RoboDK station: TECLADO.rdk

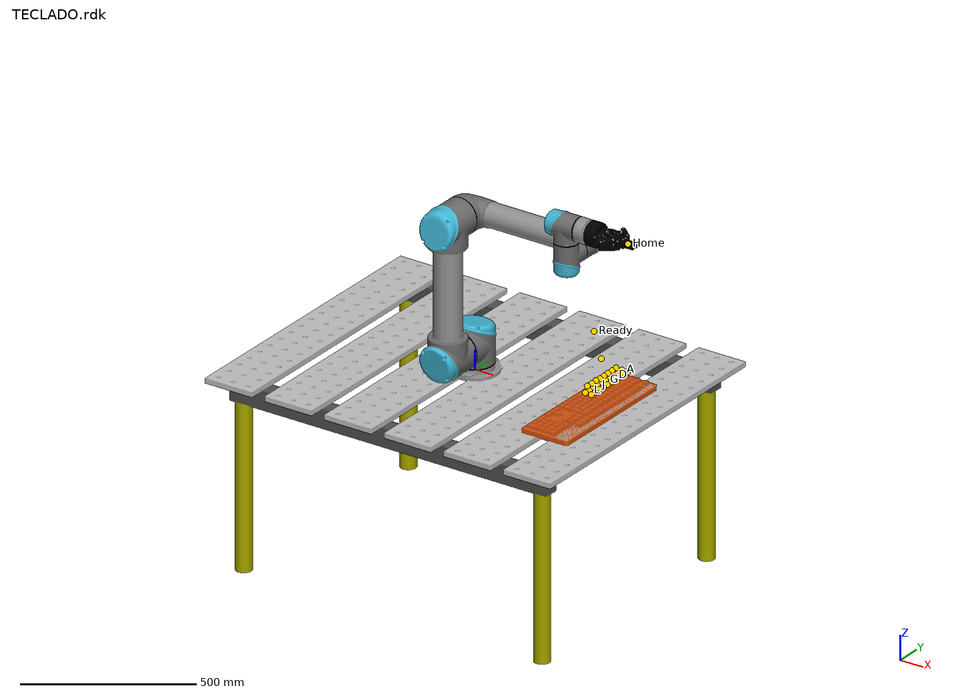
[picture v0: the station drawn from its stored meshes, robots at their saved joint values, targets as dots, program paths as lines]
Station TECLADO (saved by RoboDK 5.5.4). Poses are relative to the parent item; angles as X-Y-Z fixed-axis rotations.
  - frame UR5 Base at (0, 1000, 0) mm
    - robot UR5: 6 axes
        modified DH rows (alpha deg, a mm, theta deg, d mm): 0, 0, 0, 89.2; 90, 0, 180, 0; 0, 425, 0, 0; 0, 392, 0, 109.3; -90, 0, 0, 94.75; 90, 0, 180, 82.5
        joint limits [-360, -360, -360, -360, -360, -360] to [360, 360, 360, 360, 360, 360]; home [0, -90, -90, 0, 90, 0]; saved at [0, -90, -90, 0, 90, 0]
      - tool RobotiQ 2F-85 Gripper (Fully Closed), TCP at (0, 0, 130) mm, size 121.5 x 75 x 160.2 mm
    - object Table 1200x1000mm (Welding) at (0, 0, 0) mm, size 1193.8 x 965.2 x 609.6 mm, geometry from Table-1200x1000mm-Welding (1).sld
    - target Home (Cartesian target) at (604.5, -109.3, 608.95) mm, rotated rx -90 ry 0 rz -90 deg; joints [0, -90, -90, 0, 90, 0] of UR5
    - target Ready (Cartesian target) at (486.75, -109.3, 301.7) mm, rotated rx -180 ry 0 rz -90 deg; joints [0, -90, -90, -90, 90, 0] of UR5
    - target A (Cartesian target) at (400.33, 152.85, 49.84) mm, rotated rx -180 ry 0 rz -90 deg; joints [35.675, -92.543, -127.355, -50.102, 90, 35.675] of UR5
    - target S (Cartesian target) at (400.33, 132.85, 49.84) mm, rotated rx -180 ry 0 rz -90 deg; joints [33.377, -91.633, -128.312, -50.055, 90, 33.377] of UR5
    - target D (Cartesian target) at (400.33, 112.85, 49.84) mm, rotated rx -180 ry 0 rz -90 deg; joints [30.978, -90.828, -129.142, -50.03, 90, 30.978] of UR5
    - target F (Cartesian target) at (400.33, 92.85, 49.84) mm, rotated rx -180 ry 0 rz -90 deg; joints [28.482, -90.138, -129.84, -50.022, 90, 28.482] of UR5
    - target G (Cartesian target) at (400.33, 72.85, 49.84) mm, rotated rx -180 ry 0 rz -90 deg; joints [25.895, -89.569, -130.406, -50.024, 90, 25.895] of UR5
    - target H (Cartesian target) at (400.33, 52.85, 49.84) mm, rotated rx -180 ry 0 rz -90 deg; joints [23.225, -89.131, -130.838, -50.031, 90, 23.225] of UR5
    - target J (Cartesian target) at (400.33, 32.85, 49.84) mm, rotated rx -180 ry 0 rz -90 deg; joints [20.481, -88.828, -131.133, -50.039, 90, 20.481] of UR5
    - target K (Cartesian target) at (400.33, 12.85, 49.84) mm, rotated rx -180 ry 0 rz -90 deg; joints [17.674, -88.666, -131.29, -50.044, 90, 17.674] of UR5
    - target L (Cartesian target) at (400.33, -7.15, 49.84) mm, rotated rx -180 ry 0 rz -90 deg; joints [14.818, -88.645, -131.31, -50.044, 90, 14.818] of UR5
    - target Ñ (Cartesian target) at (400.33, -27.15, 49.84) mm, rotated rx -180 ry 0 rz -90 deg; joints [11.927, -88.768, -131.192, -50.041, 90, 11.927] of UR5
    - target Z (Cartesian target) at (380.33, 152.85, 49.84) mm, rotated rx -180 ry 0 rz -90 deg; joints [37.36, -89.989, -129.989, -50.022, 90, 37.36] of UR5
    - target X (Cartesian target) at (380.33, 132.85, 49.84) mm, rotated rx -180 ry 0 rz -90 deg; joints [34.996, -88.998, -130.968, -50.034, 90, 34.996] of UR5
    - target C (Cartesian target) at (380.33, 112.85, 49.84) mm, rotated rx -180 ry 0 rz -90 deg; joints [32.519, -88.118, -131.817, -50.066, 90, 32.519] of UR5
    - target V (Cartesian target) at (380.33, 92.85, 49.84) mm, rotated rx -180 ry 0 rz -90 deg; joints [29.93, -87.36, -132.533, -50.108, 90, 29.93] of UR5
    - target B (Cartesian target) at (380.33, 72.85, 49.84) mm, rotated rx -180 ry 0 rz -90 deg; joints [27.238, -86.734, -133.112, -50.153, 90, 27.238] of UR5
    - target N (Cartesian target) at (380.33, 52.85, 49.84) mm, rotated rx -180 ry 0 rz -90 deg; joints [24.449, -86.25, -133.555, -50.195, 90, 24.449] of UR5
    - target N (Cartesian target) at (380.33, 32.85, 49.84) mm, rotated rx -180 ry 0 rz -90 deg; joints [21.574, -85.916, -133.857, -50.227, 90, 21.574] of UR5
    - target M (Cartesian target) at (380.33, 12.85, 49.84) mm, rotated rx -180 ry 0 rz -90 deg; joints [18.626, -85.736, -134.019, -50.246, 90, 18.626] of UR5
    - target Q (Cartesian target) at (420.33, 152.85, 49.84) mm, rotated rx -180 ry 0 rz -90 deg; joints [34.128, -95.022, -124.646, -50.332, 90, 34.128] of UR5
    - target W (Cartesian target) at (420.33, 132.85, 49.84) mm, rotated rx -180 ry 0 rz -90 deg; joints [31.895, -94.18, -125.582, -50.237, 90, 31.895] of UR5
    - target E (Cartesian target) at (420.33, 112.85, 49.84) mm, rotated rx -180 ry 0 rz -90 deg; joints [29.573, -93.439, -126.393, -50.168, 90, 29.573] of UR5
    - target R (Cartesian target) at (420.33, 92.85, 49.84) mm, rotated rx -180 ry 0 rz -90 deg; joints [27.165, -92.805, -127.076, -50.119, 90, 27.165] of UR5
    - target T (Cartesian target) at (420.33, 72.85, 49.84) mm, rotated rx -180 ry 0 rz -90 deg; joints [24.678, -92.284, -127.629, -50.086, 90, 24.678] of UR5
    - target Y (Cartesian target) at (420.33, 52.85, 49.84) mm, rotated rx -180 ry 0 rz -90 deg; joints [22.118, -91.884, -128.051, -50.066, 90, 22.118] of UR5
    - target U (Cartesian target) at (420.33, 32.85, 49.84) mm, rotated rx -180 ry 0 rz -90 deg; joints [19.494, -91.608, -128.339, -50.054, 90, 19.494] of UR5
    - target I (Cartesian target) at (420.33, 12.85, 49.84) mm, rotated rx -180 ry 0 rz -90 deg; joints [16.816, -91.459, -128.492, -50.048, 90, 16.816] of UR5
    - target O (Cartesian target) at (420.33, -7.15, 49.84) mm, rotated rx -180 ry 0 rz -90 deg; joints [14.095, -91.441, -128.512, -50.047, 90, 14.095] of UR5
    - target P (Cartesian target) at (420.33, -27.15, 49.84) mm, rotated rx -180 ry 0 rz -90 deg; joints [11.344, -91.552, -128.396, -50.052, 90, 11.344] of UR5
    - target APROACH (Cartesian target) at (400.33, 52.85, 124.84) mm, rotated rx -180 ry 0 rz -90 deg; joints [23.225, -82.18, -123.993, -63.827, 90, 23.225] of UR5
  - Python program Prog1 (listed below)
  - object Teclado HP at (340, 1190, 0) mm, rotated rx 90 ry 0 rz -90 deg, size 450 x 25 x 160 mm, geometry from Teclado HP.stp

--- Python program Prog1 ---
# Type help("robodk.robolink") or help("robodk.robomath") for more information
# Press F5 to run the script
# Documentation: https://robodk.com/doc/en/RoboDK-API.html
# Reference:     https://robodk.com/doc/en/PythonAPI/robodk.html
# Note: It is not required to keep a copy of this file, your Python script is saved with your RDK project

# You can also use the new version of the API:
from robodk import robolink    # RoboDK API
from robodk import robomath    # Robot toolbox
RDK = robolink.Robolink()

# Forward and backwards compatible use of the RoboDK API:
# Remove these 2 lines to follow python programming guidelines
from robodk import *      # RoboDK API
from robolink import *    # Robot toolbox
# Link to RoboDK
# RDK = Robolink()

RDK = Robolink() # establish a link with the simulator
robot = RDK.Item('UR5')      # retrieve the robot by name

# Program example:
item = RDK.Item('base')
if item.Valid():
    print('Item selected: ' + item.Name())
    print('Item posistion: ' + repr(item.Pose()))

print('Items in the station:')
itemlist = RDK.ItemList()
print(itemlist)

home = RDK.Item('Home')         # retrieve the Target item
robot.MoveJ(home)                 # move the robot to the target

ready = RDK.Item('Ready')
robot.MoveJ(ready)               # linear move to the approach position

ins_call = mbox("Enter a program call to add after each movement", entry = "SynchRobot")

for caracter in ins_call:
    if caracter.isalpha():
        target = RDK.Item(caracter.upper())
        approach = target.Pose()*transl(0,0,-100)
        robot.MoveJ(approach)               # linear move to the approach position
        time.sleep(1)
        robot.MoveL(target)
        time.sleep(1)
        robot.MoveL(approach)

robot.MoveJ(ready)               # linear move to the approach position
robot.MoveJ(home)                 # move the robot to the target
